// Mitsubishi GX Works2 project: C412_23-08-19 Backup   PLC: Q03UDE

PROGRAM MAIN
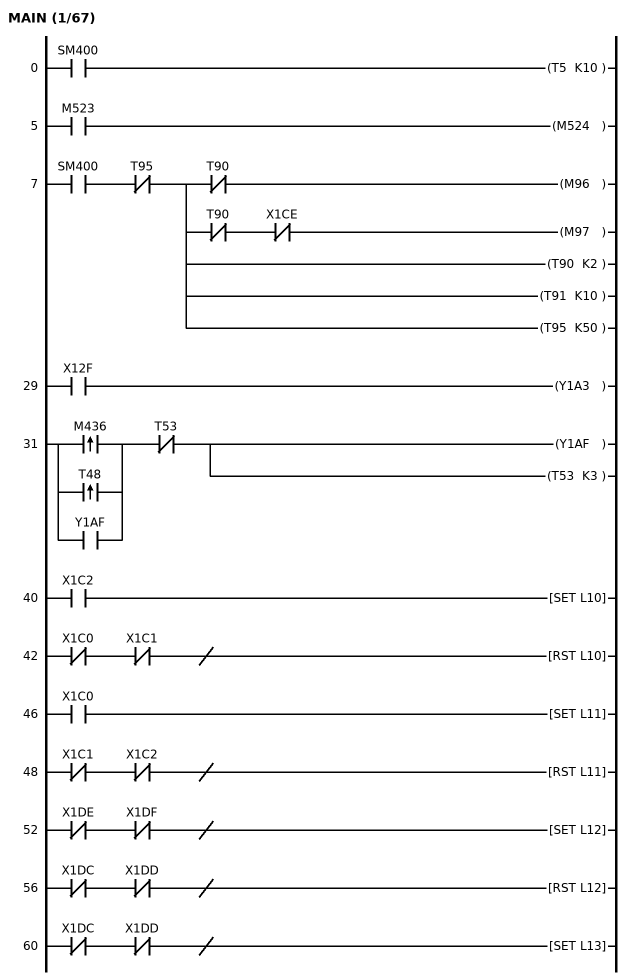
0     LD      SM400
      OUT     T5 K10
5     LD      M523
      OUT     M524
7     LD      SM400
      ANI     T95
      MPS
      ANI     T90
      OUT     M96
      MRD
      ANI     T90
      ANI     X1CE
      OUT     M97
      MPP
      OUT     T90 K2
      OUT     T91 K10
      OUT     T95 K50
29    LD      X12F
      OUT     Y1A3
31    LDP     M436
      ORP     T48
      OR      Y1AF
      ANI     T53
      OUT     Y1AF
      OUT     T53 K3
40    LD      X1C2
      SET     L10
42    LDI     X1C0
      ANI     X1C1
      INV
      RST     L10
46    LD      X1C0
      SET     L11
48    LDI     X1C1
      ANI     X1C2
      INV
      RST     L11
52    LDI     X1DE
      ANI     X1DF
      INV
      SET     L12
56    LDI     X1DC
      ANI     X1DD
      INV
      RST     L12
60    LDI     X1DC
      ANI     X1DD
      INV
      SET     L13
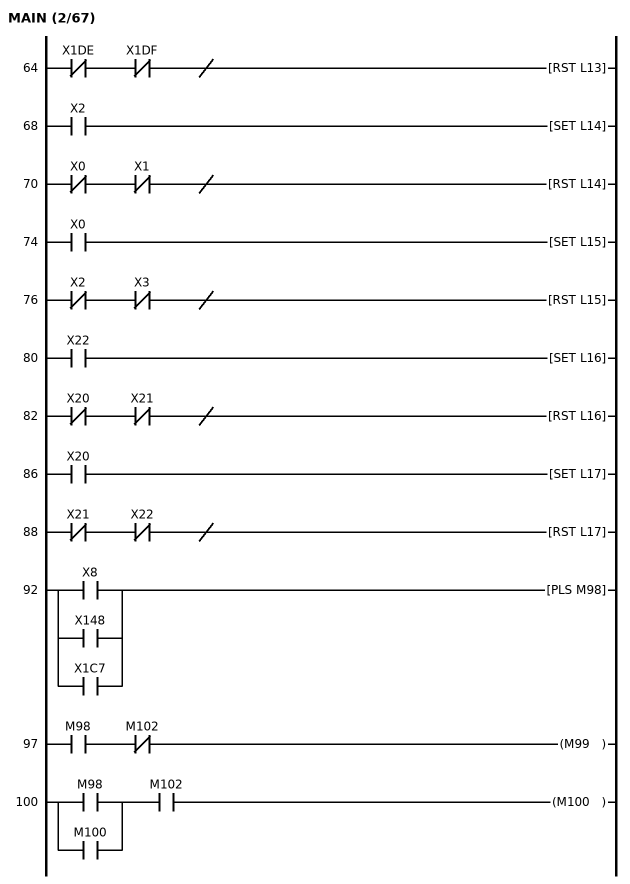
64    LDI     X1DE
      ANI     X1DF
      INV
      RST     L13
68    LD      X2
      SET     L14
70    LDI     X0
      ANI     X1
      INV
      RST     L14
74    LD      X0
      SET     L15
76    LDI     X2
      ANI     X3
      INV
      RST     L15
80    LD      X22
      SET     L16
82    LDI     X20
      ANI     X21
      INV
      RST     L16
86    LD      X20
      SET     L17
88    LDI     X21
      ANI     X22
      INV
      RST     L17
92    LD      X8
      OR      X148
      OR      X1C7
      PLS     M98
97    LD      M98
      ANI     M102
      OUT     M99
100   LD      M98
      OR      M100
      AND     M102
      OUT     M100
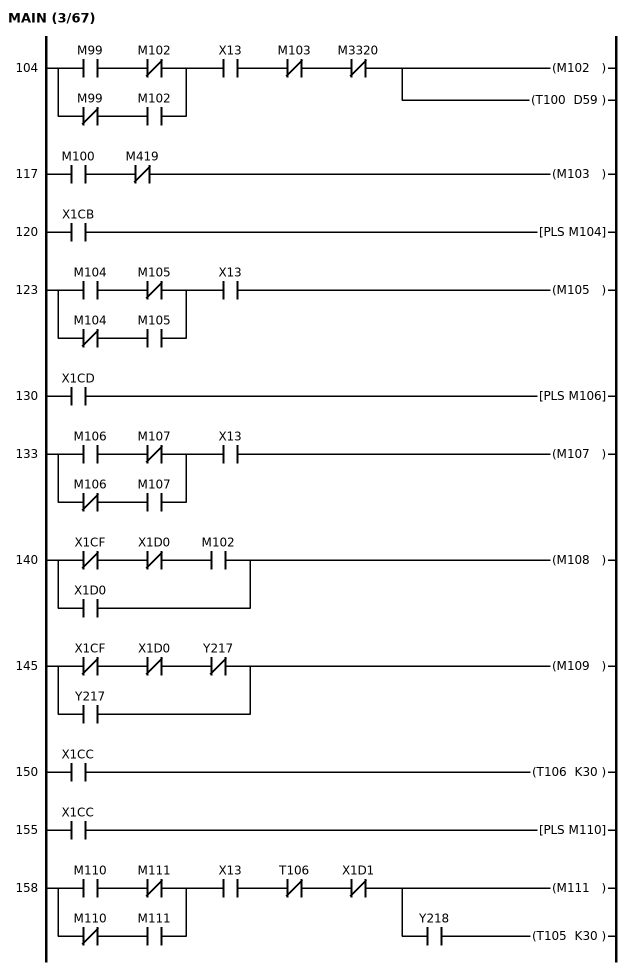
104   LD      M99
      ANI     M102
      LDI     M99
      AND     M102
      ORB
      AND     X13
      ANI     M103
      ANI     M3320
      OUT     M102
      OUT     T100 D59
117   LD      M100
      ANI     M419
      OUT     M103
120   LD      X1CB
      PLS     M104
123   LD      M104
      ANI     M105
      LDI     M104
      AND     M105
      ORB
      AND     X13
      OUT     M105
130   LD      X1CD
      PLS     M106
133   LD      M106
      ANI     M107
      LDI     M106
      AND     M107
      ORB
      AND     X13
      OUT     M107
140   LDI     X1CF
      ANI     X1D0
      AND     M102
      OR      X1D0
      OUT     M108
145   LDI     X1CF
      ANI     X1D0
      ANI     Y217
      OR      Y217
      OUT     M109
150   LD      X1CC
      OUT     T106 K30
155   LD      X1CC
      PLS     M110
158   LD      M110
      ANI     M111
      LDI     M110
      AND     M111
      ORB
      AND     X13
      ANI     T106
      ANI     X1D1
      OUT     M111
      AND     Y218
      OUT     T105 K30
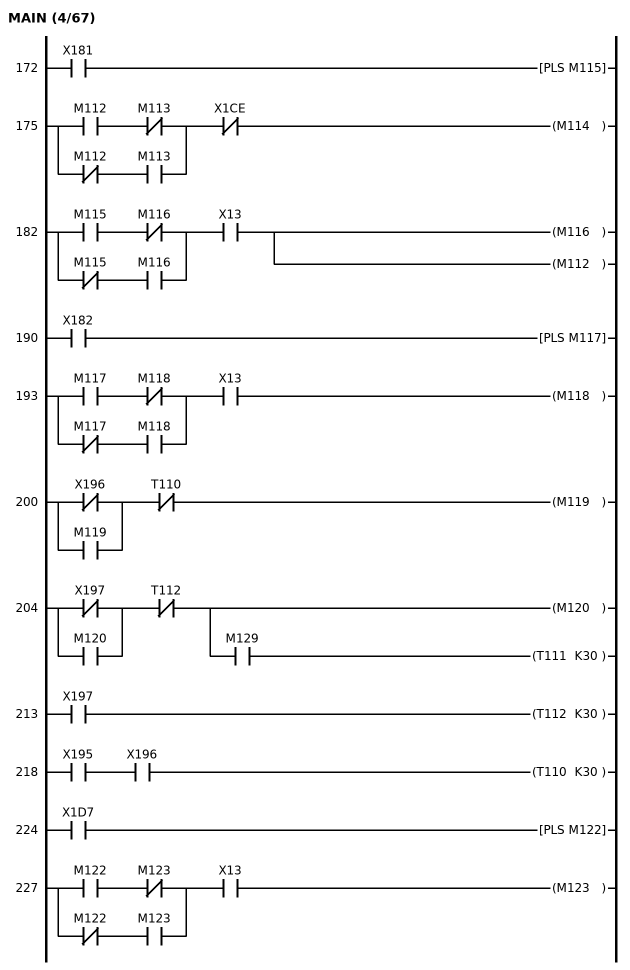
172   LD      X181
      PLS     M115
175   LD      M112
      ANI     M113
      LDI     M112
      AND     M113
      ORB
      ANI     X1CE
      OUT     M114
182   LD      M115
      ANI     M116
      LDI     M115
      AND     M116
      ORB
      AND     X13
      OUT     M116
      OUT     M112
190   LD      X182
      PLS     M117
193   LD      M117
      ANI     M118
      LDI     M117
      AND     M118
      ORB
      AND     X13
      OUT     M118
200   LDI     X196
      OR      M119
      ANI     T110
      OUT     M119
204   LDI     X197
      OR      M120
      ANI     T112
      OUT     M120
      AND     M129
      OUT     T111 K30
213   LD      X197
      OUT     T112 K30
218   LD      X195
      AND     X196
      OUT     T110 K30
224   LD      X1D7
      PLS     M122
227   LD      M122
      ANI     M123
      LDI     M122
      AND     M123
      ORB
      AND     X13
      OUT     M123
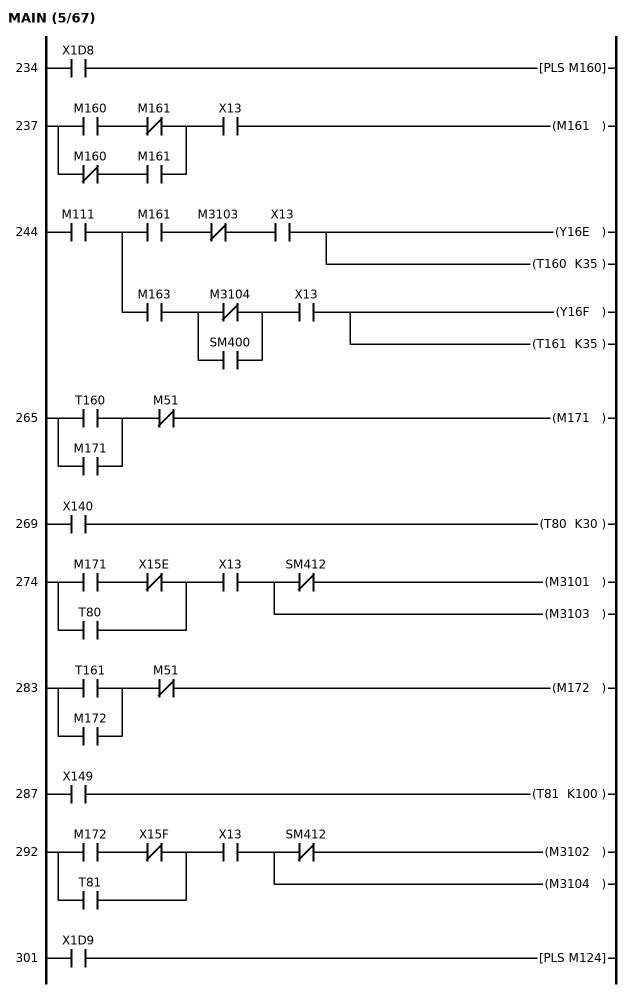
234   LD      X1D8
      PLS     M160
237   LD      M160
      ANI     M161
      LDI     M160
      AND     M161
      ORB
      AND     X13
      OUT     M161
244   LD      M111
      MPS
      AND     M161
      ANI     M3103
      AND     X13
      OUT     Y16E
      OUT     T160 K35
      MPP
      AND     M163
      LDI     M3104
      OR      SM400
      ANB
      AND     X13
      OUT     Y16F
      OUT     T161 K35
265   LD      T160
      OR      M171
      ANI     M51
      OUT     M171
269   LD      X140
      OUT     T80 K30
274   LD      M171
      ANI     X15E
      OR      T80
      AND     X13
      MPS
      ANI     SM412
      OUT     M3101
      MPP
      OUT     M3103
283   LD      T161
      OR      M172
      ANI     M51
      OUT     M172
287   LD      X149
      OUT     T81 K100
292   LD      M172
      ANI     X15F
      OR      T81
      AND     X13
      MPS
      ANI     SM412
      OUT     M3102
      MPP
      OUT     M3104
301   LD      X1D9
      PLS     M124
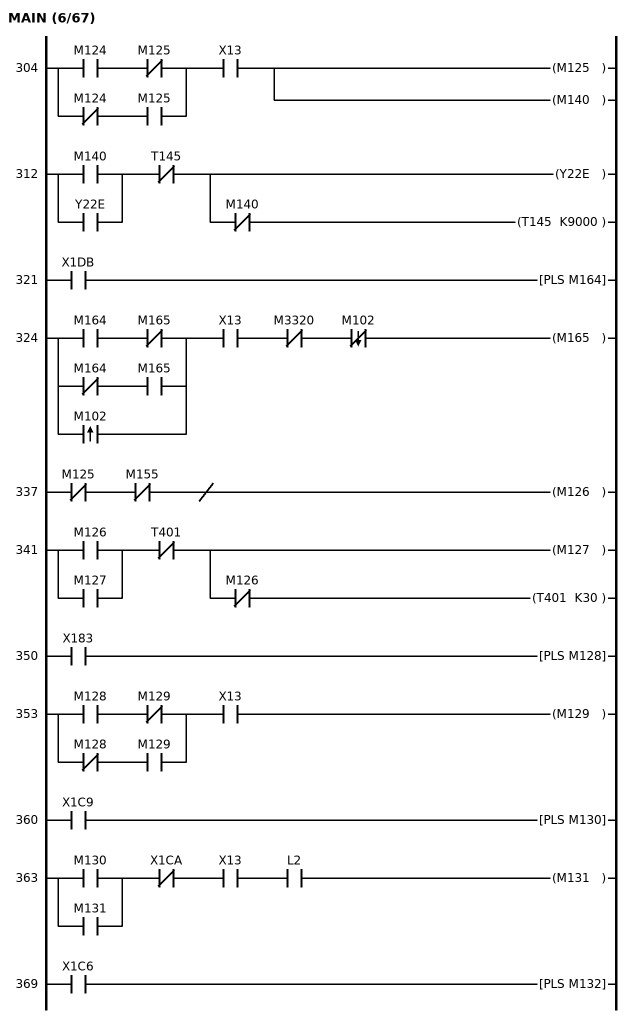
304   LD      M124
      ANI     M125
      LDI     M124
      AND     M125
      ORB
      AND     X13
      OUT     M125
      OUT     M140
312   LD      M140
      OR      Y22E
      ANI     T145
      OUT     Y22E
      ANI     M140
      OUT     T145 K9000
321   LD      X1DB
      PLS     M164
324   LD      M164
      ANI     M165
      LDI     M164
      AND     M165
      ORB
      ORP     M102
      AND     X13
      ANI     M3320
      ANDFI   M102
      OUT     M165
337   LDI     M125
      ANI     M155
      INV
      OUT     M126
341   LD      M126
      OR      M127
      ANI     T401
      OUT     M127
      ANI     M126
      OUT     T401 K30
350   LD      X183
      PLS     M128
353   LD      M128
      ANI     M129
      LDI     M128
      AND     M129
      ORB
      AND     X13
      OUT     M129
360   LD      X1C9
      PLS     M130
363   LD      M130
      OR      M131
      ANI     X1CA
      AND     X13
      AND     L2
      OUT     M131
369   LD      X1C6
      PLS     M132
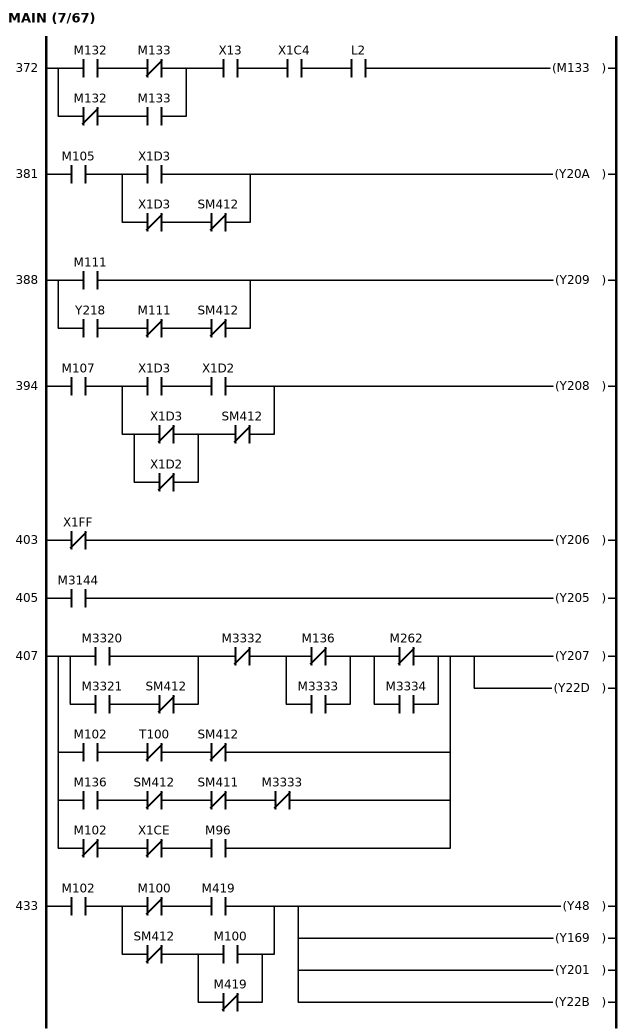
372   LD      M132
      ANI     M133
      LDI     M132
      AND     M133
      ORB
      AND     X13
      AND     X1C4
      AND     L2
      OUT     M133
381   LD      M105
      LD      X1D3
      LDI     X1D3
      ANI     SM412
      ORB
      ANB
      OUT     Y20A
388   LD      M111
      LD      Y218
      ANI     M111
      ANI     SM412
      ORB
      OUT     Y209
394   LD      M107
      LD      X1D3
      AND     X1D2
      LDI     X1D3
      ORI     X1D2
      ANI     SM412
      ORB
      ANB
      OUT     Y208
403   LDI     X1FF
      OUT     Y206
405   LD      M3144
      OUT     Y205
407   LD      M3320
      LD      M3321
      ANI     SM412
      ORB
      ANI     M3332
      LDI     M136
      OR      M3333
      ANB
      LDI     M262
      OR      M3334
      ANB
      LD      M102
      ANI     T100
      ANI     SM412
      ORB
      LD      M136
      ANI     SM412
      ANI     SM411
      ANI     M3333
      ORB
      LDI     M102
      ANI     X1CE
      AND     M96
      ORB
      OUT     Y207
      OUT     Y22D
433   LD      M102
      LDI     M100
      AND     M419
      LDI     SM412
      LD      M100
      ORI     M419
      ANB
      ORB
      ANB
      OUT     Y48
      OUT     Y169
      OUT     Y201
      OUT     Y22B
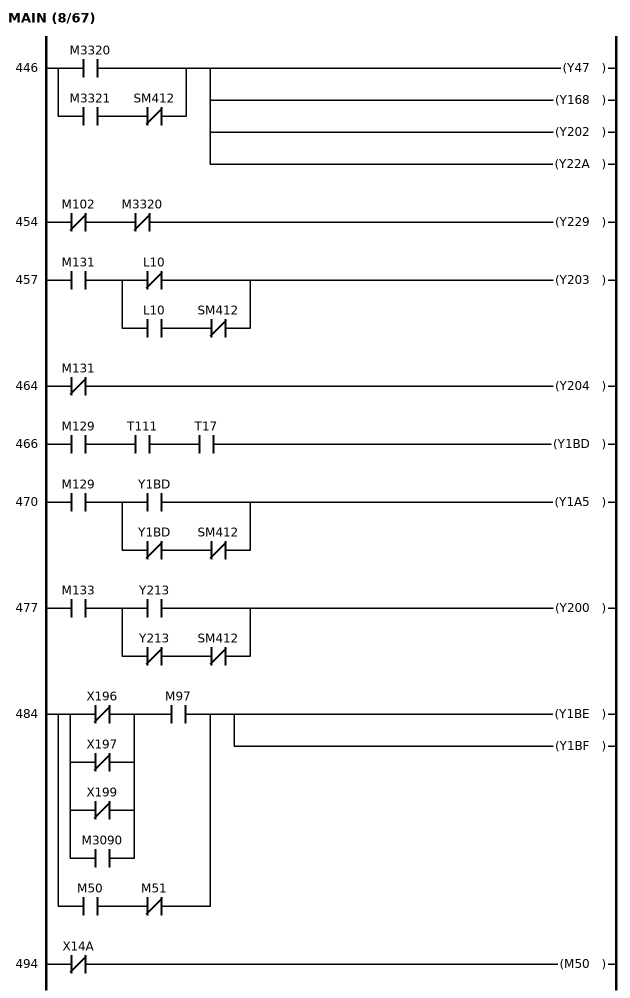
446   LD      M3320
      LD      M3321
      ANI     SM412
      ORB
      OUT     Y47
      OUT     Y168
      OUT     Y202
      OUT     Y22A
454   LDI     M102
      ANI     M3320
      OUT     Y229
457   LD      M131
      LDI     L10
      LD      L10
      ANI     SM412
      ORB
      ANB
      OUT     Y203
464   LDI     M131
      OUT     Y204
466   LD      M129
      AND     T111
      AND     T17
      OUT     Y1BD
470   LD      M129
      LD      Y1BD
      LDI     Y1BD
      ANI     SM412
      ORB
      ANB
      OUT     Y1A5
477   LD      M133
      LD      Y213
      LDI     Y213
      ANI     SM412
      ORB
      ANB
      OUT     Y200
484   LDI     X196
      ORI     X197
      ORI     X199
      OR      M3090
      AND     M97
      LD      M50
      ANI     M51
      ORB
      OUT     Y1BE
      OUT     Y1BF
494   LDI     X14A
      OUT     M50
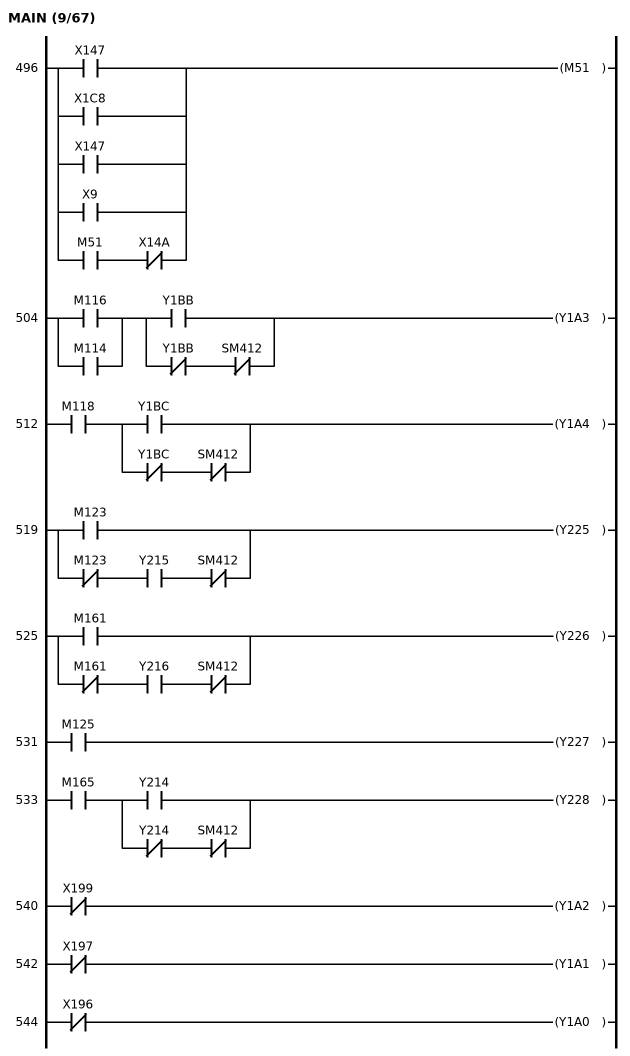
496   LD      X147
      OR      X1C8
      OR      X147
      OR      X9
      LD      M51
      ANI     X14A
      ORB
      OUT     M51
504   LD      M116
      OR      M114
      LD      Y1BB
      LDI     Y1BB
      ANI     SM412
      ORB
      ANB
      OUT     Y1A3
512   LD      M118
      LD      Y1BC
      LDI     Y1BC
      ANI     SM412
      ORB
      ANB
      OUT     Y1A4
519   LD      M123
      LDI     M123
      AND     Y215
      ANI     SM412
      ORB
      OUT     Y225
525   LD      M161
      LDI     M161
      AND     Y216
      ANI     SM412
      ORB
      OUT     Y226
531   LD      M125
      OUT     Y227
533   LD      M165
      LD      Y214
      LDI     Y214
      ANI     SM412
      ORB
      ANB
      OUT     Y228
540   LDI     X199
      OUT     Y1A2
542   LDI     X197
      OUT     Y1A1
544   LDI     X196
      OUT     Y1A0
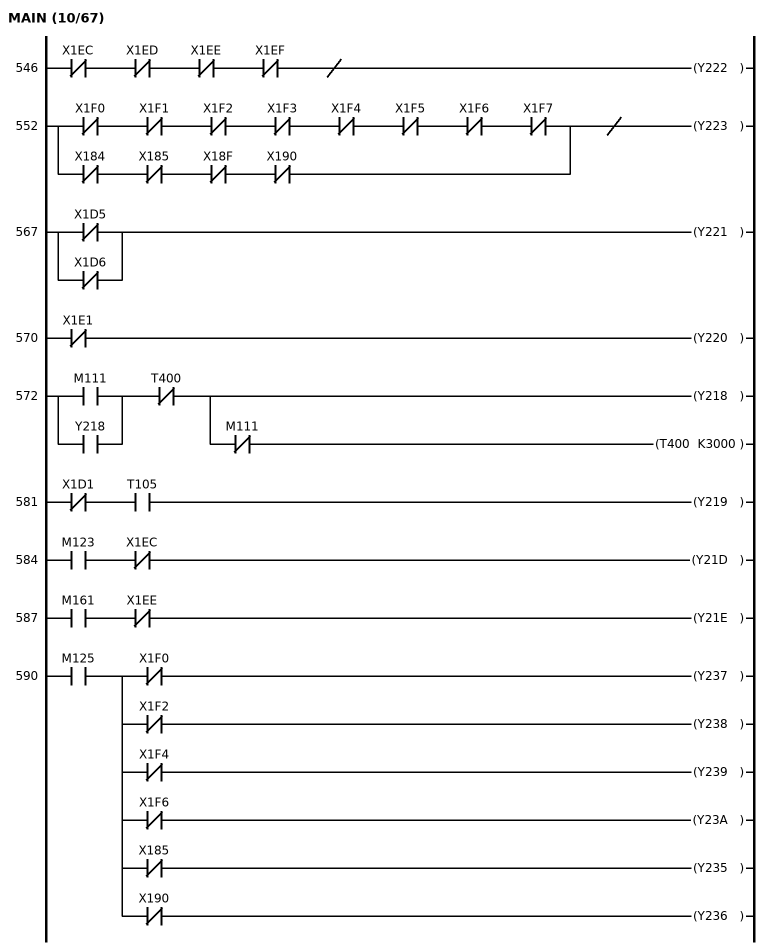
546   LDI     X1EC
      ANI     X1ED
      ANI     X1EE
      ANI     X1EF
      INV
      OUT     Y222
552   LDI     X1F0
      ANI     X1F1
      ANI     X1F2
      ANI     X1F3
      ANI     X1F4
      ANI     X1F5
      ANI     X1F6
      ANI     X1F7
      LDI     X184
      ANI     X185
      ANI     X18F
      ANI     X190
      ORB
      INV
      OUT     Y223
567   LDI     X1D5
      ORI     X1D6
      OUT     Y221
570   LDI     X1E1
      OUT     Y220
572   LD      M111
      OR      Y218
      ANI     T400
      OUT     Y218
      ANI     M111
      OUT     T400 K3000
581   LDI     X1D1
      AND     T105
      OUT     Y219
584   LD      M123
      ANI     X1EC
      OUT     Y21D
587   LD      M161
      ANI     X1EE
      OUT     Y21E
590   LD      M125
      MPS
      ANI     X1F0
      OUT     Y237
      MRD
      ANI     X1F2
      OUT     Y238
      MRD
      ANI     X1F4
      OUT     Y239
      MRD
      ANI     X1F6
      OUT     Y23A
      MRD
      ANI     X185
      OUT     Y235
      MPP
      ANI     X190
      OUT     Y236
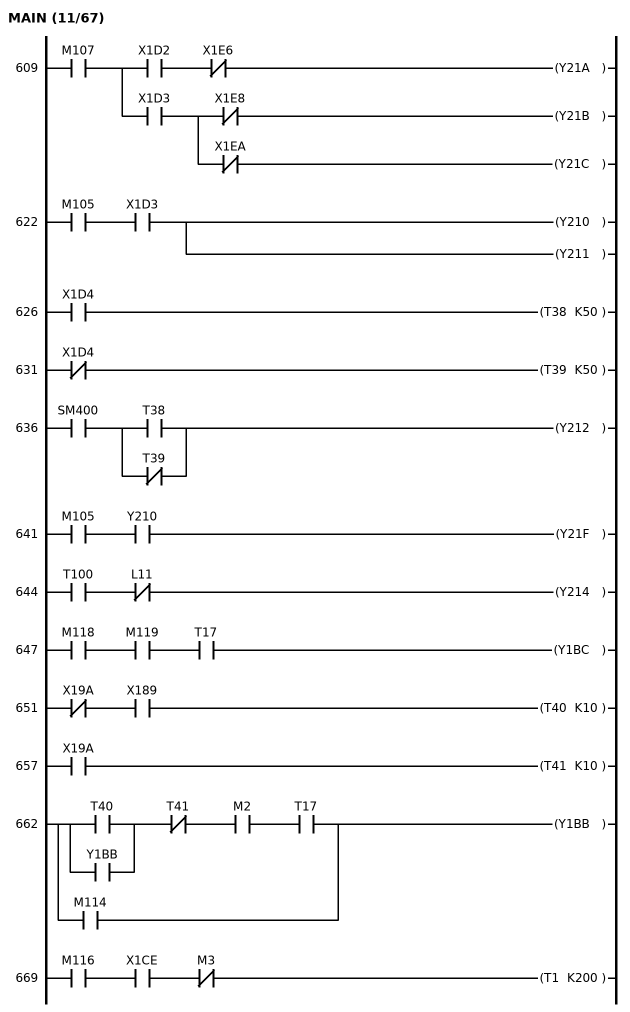
609   LD      M107
      MPS
      AND     X1D2
      ANI     X1E6
      OUT     Y21A
      MPP
      AND     X1D3
      MPS
      ANI     X1E8
      OUT     Y21B
      MPP
      ANI     X1EA
      OUT     Y21C
622   LD      M105
      AND     X1D3
      OUT     Y210
      OUT     Y211
626   LD      X1D4
      OUT     T38 K50
631   LDI     X1D4
      OUT     T39 K50
636   LD      SM400
      LD      T38
      ORI     T39
      ANB
      OUT     Y212
641   LD      M105
      AND     Y210
      OUT     Y21F
644   LD      T100
      ANI     L11
      OUT     Y214
647   LD      M118
      AND     M119
      AND     T17
      OUT     Y1BC
651   LDI     X19A
      AND     X189
      OUT     T40 K10
657   LD      X19A
      OUT     T41 K10
662   LD      T40
      OR      Y1BB
      ANI     T41
      AND     M2
      AND     T17
      OR      M114
      OUT     Y1BB
669   LD      M116
      AND     X1CE
      ANI     M3
      OUT     T1 K200
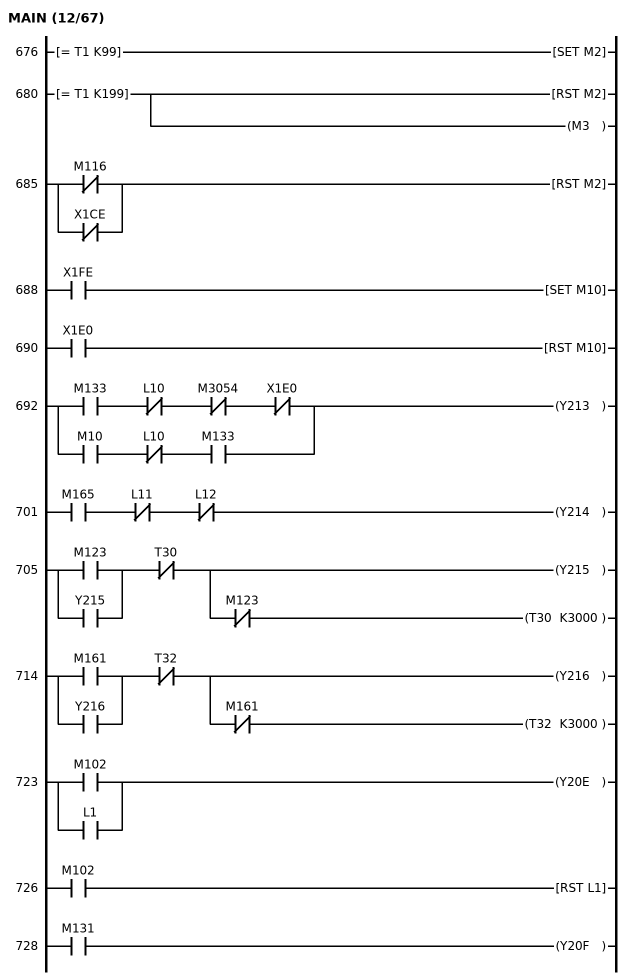
676   LD=     T1 K99
      SET     M2
680   LD=     T1 K199
      RST     M2
      OUT     M3
685   LDI     M116
      ORI     X1CE
      RST     M2
688   LD      X1FE
      SET     M10
690   LD      X1E0
      RST     M10
692   LD      M133
      ANI     L10
      ANI     M3054
      ANI     X1E0
      LD      M10
      ANI     L10
      AND     M133
      ORB
      OUT     Y213
701   LD      M165
      ANI     L11
      ANI     L12
      OUT     Y214
705   LD      M123
      OR      Y215
      ANI     T30
      OUT     Y215
      ANI     M123
      OUT     T30 K3000
714   LD      M161
      OR      Y216
      ANI     T32
      OUT     Y216
      ANI     M161
      OUT     T32 K3000
723   LD      M102
      OR      L1
      OUT     Y20E
726   LD      M102
      RST     L1
728   LD      M131
      OUT     Y20F
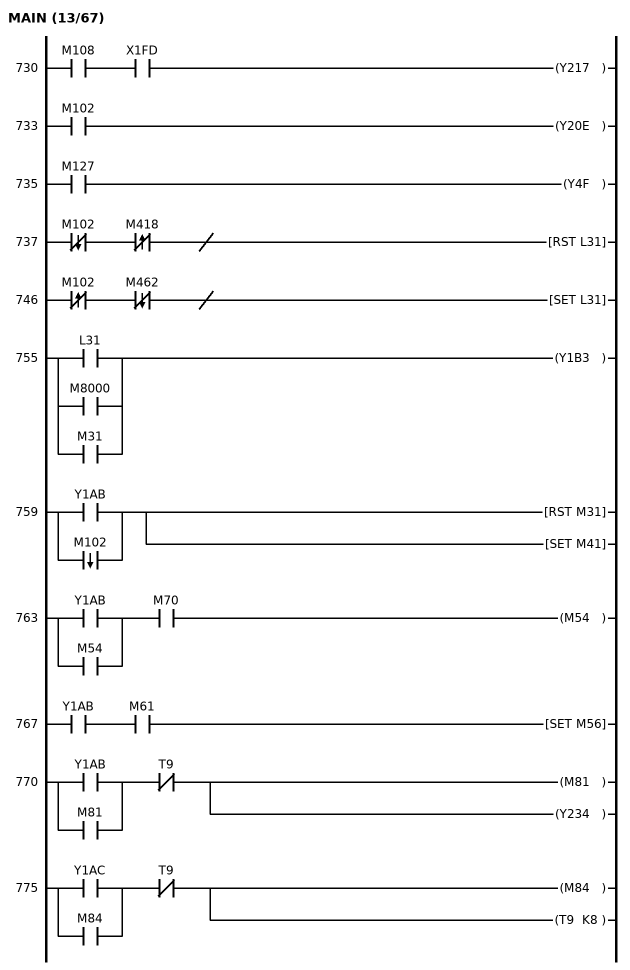
730   LD      M108
      AND     X1FD
      OUT     Y217
733   LD      M102
      OUT     Y20E
735   LD      M127
      OUT     Y4F
737   LDFI    M102
      ANDPI   M418
      INV
      RST     L31
746   LDPI    M102
      ANDFI   M462
      INV
      SET     L31
755   LD      L31
      OR      M8000
      OR      M31
      OUT     Y1B3
759   LD      Y1AB
      ORF     M102
      RST     M31
      SET     M41
763   LD      Y1AB
      OR      M54
      AND     M70
      OUT     M54
767   LD      Y1AB
      AND     M61
      SET     M56
770   LD      Y1AB
      OR      M81
      ANI     T9
      OUT     M81
      OUT     Y234
775   LD      Y1AC
      OR      M84
      ANI     T9
      OUT     M84
      OUT     T9 K8
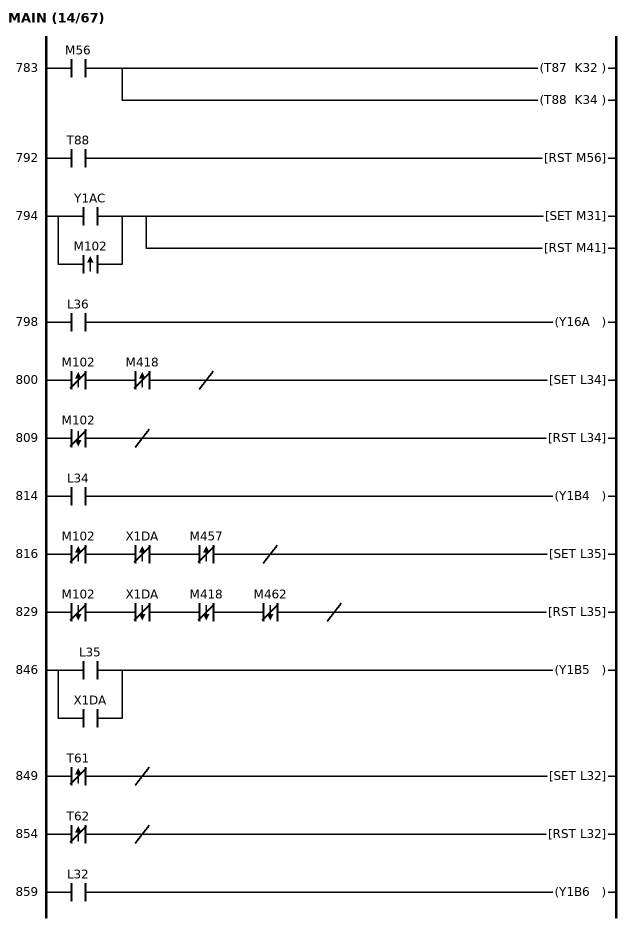
783   LD      M56
      OUT     T87 K32
      OUT     T88 K34
792   LD      T88
      RST     M56
794   LD      Y1AC
      ORP     M102
      SET     M31
      RST     M41
798   LD      L36
      OUT     Y16A
800   LDPI    M102
      ANDPI   M418
      INV
      SET     L34
809   LDFI    M102
      INV
      RST     L34
814   LD      L34
      OUT     Y1B4
816   LDPI    M102
      ANDPI   X1DA
      ANDPI   M457
      INV
      SET     L35
829   LDFI    M102
      ANDFI   X1DA
      ANDFI   M418
      ANDFI   M462
      INV
      RST     L35
846   LD      L35
      OR      X1DA
      OUT     Y1B5
849   LDPI    T61
      INV
      SET     L32
854   LDPI    T62
      INV
      RST     L32
859   LD      L32
      OUT     Y1B6
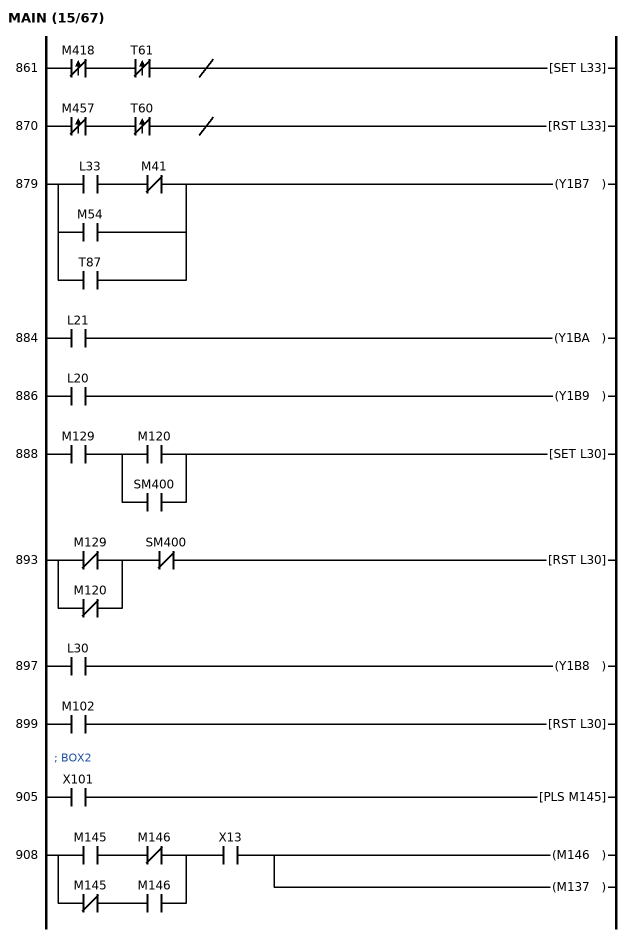
861   LDPI    M418
      ANDPI   T61
      INV
      SET     L33
870   LDPI    M457
      ANDPI   T60
      INV
      RST     L33
879   LD      L33
      ANI     M41
      OR      M54
      OR      T87
      OUT     Y1B7
884   LD      L21
      OUT     Y1BA
886   LD      L20
      OUT     Y1B9
888   LD      M129
      LD      M120
      OR      SM400
      ANB
      SET     L30
893   LDI     M129
      ORI     M120
      ANI     SM400
      RST     L30
897   LD      L30
      OUT     Y1B8
899   LD      M102
      RST     L30
; BOX2
905   LD      X101
      PLS     M145
908   LD      M145
      ANI     M146
      LDI     M145
      AND     M146
      ORB
      AND     X13
      OUT     M146
      OUT     M137
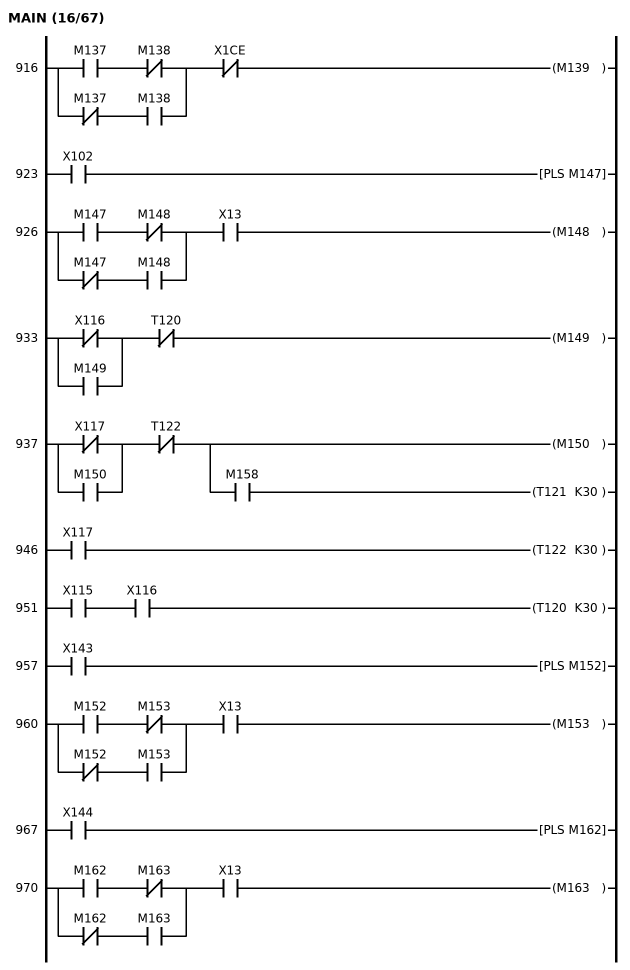
916   LD      M137
      ANI     M138
      LDI     M137
      AND     M138
      ORB
      ANI     X1CE
      OUT     M139
923   LD      X102
      PLS     M147
926   LD      M147
      ANI     M148
      LDI     M147
      AND     M148
      ORB
      AND     X13
      OUT     M148
933   LDI     X116
      OR      M149
      ANI     T120
      OUT     M149
937   LDI     X117
      OR      M150
      ANI     T122
      OUT     M150
      AND     M158
      OUT     T121 K30
946   LD      X117
      OUT     T122 K30
951   LD      X115
      AND     X116
      OUT     T120 K30
957   LD      X143
      PLS     M152
960   LD      M152
      ANI     M153
      LDI     M152
      AND     M153
      ORB
      AND     X13
      OUT     M153
967   LD      X144
      PLS     M162
970   LD      M162
      ANI     M163
      LDI     M162
      AND     M163
      ORB
      AND     X13
      OUT     M163
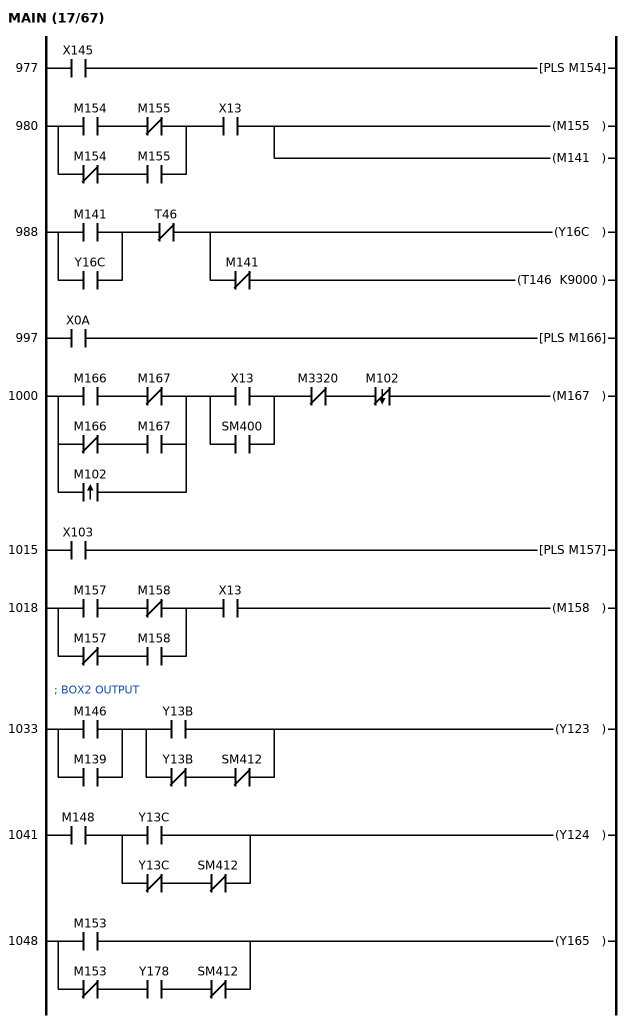
977   LD      X145
      PLS     M154
980   LD      M154
      ANI     M155
      LDI     M154
      AND     M155
      ORB
      AND     X13
      OUT     M155
      OUT     M141
988   LD      M141
      OR      Y16C
      ANI     T46
      OUT     Y16C
      ANI     M141
      OUT     T146 K9000
997   LD      X0A
      PLS     M166
1000  LD      M166
      ANI     M167
      LDI     M166
      AND     M167
      ORB
      ORP     M102
      LD      X13
      OR      SM400
      ANB
      ANI     M3320
      ANDFI   M102
      OUT     M167
1015  LD      X103
      PLS     M157
1018  LD      M157
      ANI     M158
      LDI     M157
      AND     M158
      ORB
      AND     X13
      OUT     M158
; BOX2 OUTPUT
1033  LD      M146
      OR      M139
      LD      Y13B
      LDI     Y13B
      ANI     SM412
      ORB
      ANB
      OUT     Y123
1041  LD      M148
      LD      Y13C
      LDI     Y13C
      ANI     SM412
      ORB
      ANB
      OUT     Y124
1048  LD      M153
      LDI     M153
      AND     Y178
      ANI     SM412
      ORB
      OUT     Y165
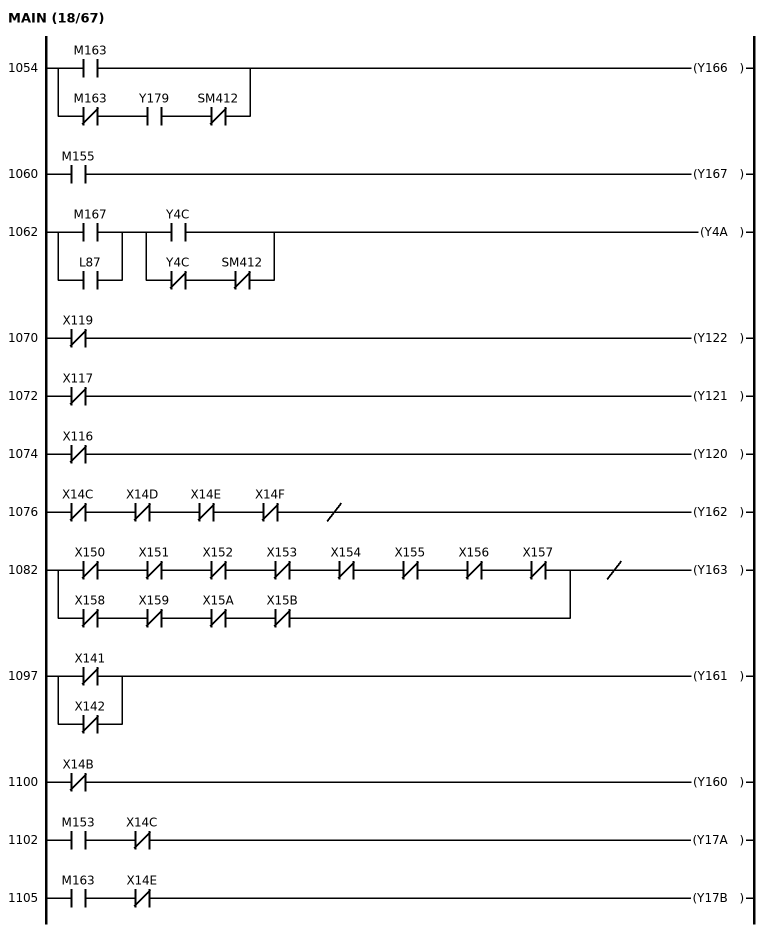
1054  LD      M163
      LDI     M163
      AND     Y179
      ANI     SM412
      ORB
      OUT     Y166
1060  LD      M155
      OUT     Y167
1062  LD      M167
      OR      L87
      LD      Y4C
      LDI     Y4C
      ANI     SM412
      ORB
      ANB
      OUT     Y4A
1070  LDI     X119
      OUT     Y122
1072  LDI     X117
      OUT     Y121
1074  LDI     X116
      OUT     Y120
1076  LDI     X14C
      ANI     X14D
      ANI     X14E
      ANI     X14F
      INV
      OUT     Y162
1082  LDI     X150
      ANI     X151
      ANI     X152
      ANI     X153
      ANI     X154
      ANI     X155
      ANI     X156
      ANI     X157
      LDI     X158
      ANI     X159
      ANI     X15A
      ANI     X15B
      ORB
      INV
      OUT     Y163
1097  LDI     X141
      ORI     X142
      OUT     Y161
1100  LDI     X14B
      OUT     Y160
1102  LD      M153
      ANI     X14C
      OUT     Y17A
1105  LD      M163
      ANI     X14E
      OUT     Y17B
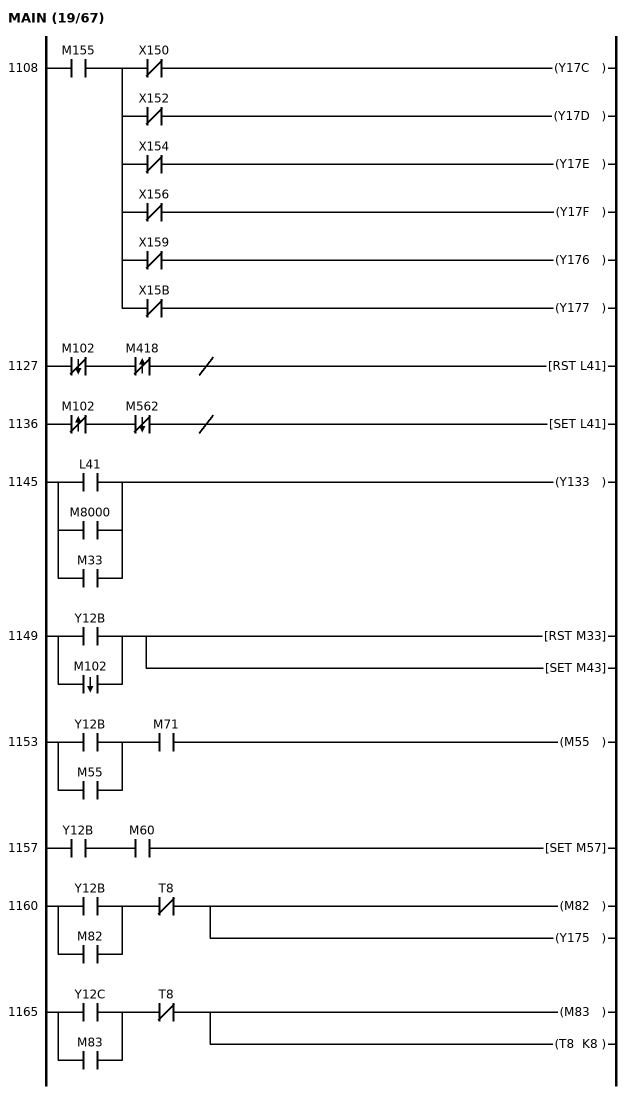
1108  LD      M155
      MPS
      ANI     X150
      OUT     Y17C
      MRD
      ANI     X152
      OUT     Y17D
      MRD
      ANI     X154
      OUT     Y17E
      MRD
      ANI     X156
      OUT     Y17F
      MRD
      ANI     X159
      OUT     Y176
      MPP
      ANI     X15B
      OUT     Y177
1127  LDFI    M102
      ANDPI   M418
      INV
      RST     L41
1136  LDPI    M102
      ANDFI   M562
      INV
      SET     L41
1145  LD      L41
      OR      M8000
      OR      M33
      OUT     Y133
1149  LD      Y12B
      ORF     M102
      RST     M33
      SET     M43
1153  LD      Y12B
      OR      M55
      AND     M71
      OUT     M55
1157  LD      Y12B
      AND     M60
      SET     M57
1160  LD      Y12B
      OR      M82
      ANI     T8
      OUT     M82
      OUT     Y175
1165  LD      Y12C
      OR      M83
      ANI     T8
      OUT     M83
      OUT     T8 K8
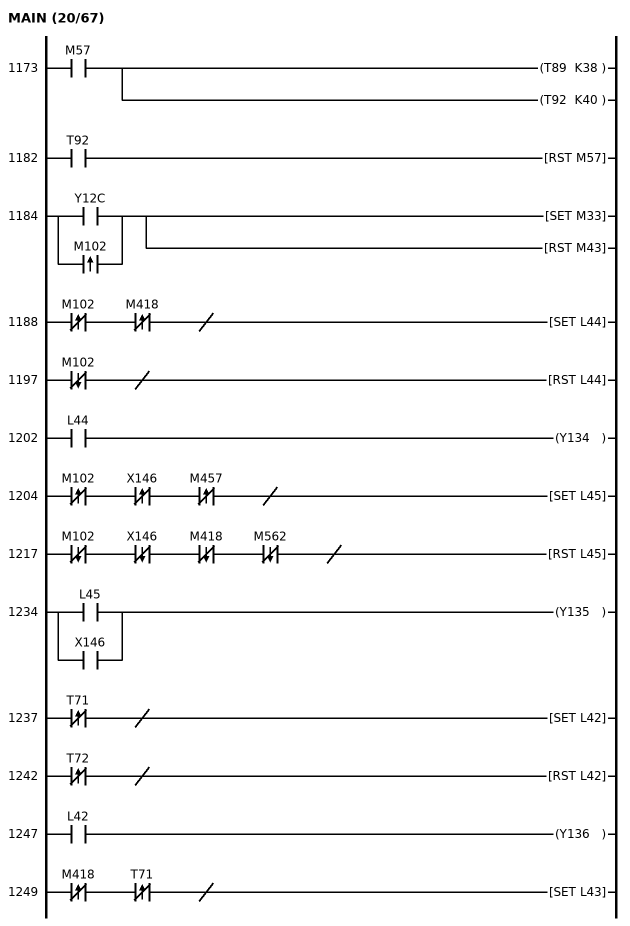
1173  LD      M57
      OUT     T89 K38
      OUT     T92 K40
1182  LD      T92
      RST     M57
1184  LD      Y12C
      ORP     M102
      SET     M33
      RST     M43
1188  LDPI    M102
      ANDPI   M418
      INV
      SET     L44
1197  LDFI    M102
      INV
      RST     L44
1202  LD      L44
      OUT     Y134
1204  LDPI    M102
      ANDPI   X146
      ANDPI   M457
      INV
      SET     L45
1217  LDFI    M102
      ANDFI   X146
      ANDFI   M418
      ANDFI   M562
      INV
      RST     L45
1234  LD      L45
      OR      X146
      OUT     Y135
1237  LDPI    T71
      INV
      SET     L42
1242  LDPI    T72
      INV
      RST     L42
1247  LD      L42
      OUT     Y136
1249  LDPI    M418
      ANDPI   T71
      INV
      SET     L43
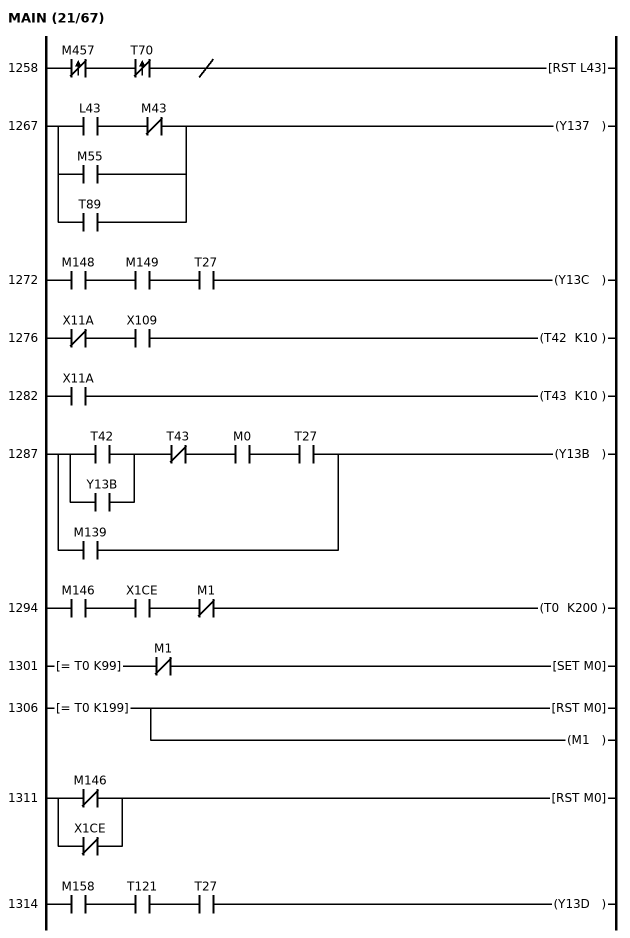
1258  LDPI    M457
      ANDPI   T70
      INV
      RST     L43
1267  LD      L43
      ANI     M43
      OR      M55
      OR      T89
      OUT     Y137
1272  LD      M148
      AND     M149
      AND     T27
      OUT     Y13C
1276  LDI     X11A
      AND     X109
      OUT     T42 K10
1282  LD      X11A
      OUT     T43 K10
1287  LD      T42
      OR      Y13B
      ANI     T43
      AND     M0
      AND     T27
      OR      M139
      OUT     Y13B
1294  LD      M146
      AND     X1CE
      ANI     M1
      OUT     T0 K200
1301  LD=     T0 K99
      ANI     M1
      SET     M0
1306  LD=     T0 K199
      RST     M0
      OUT     M1
1311  LDI     M146
      ORI     X1CE
      RST     M0
1314  LD      M158
      AND     T121
      AND     T27
      OUT     Y13D
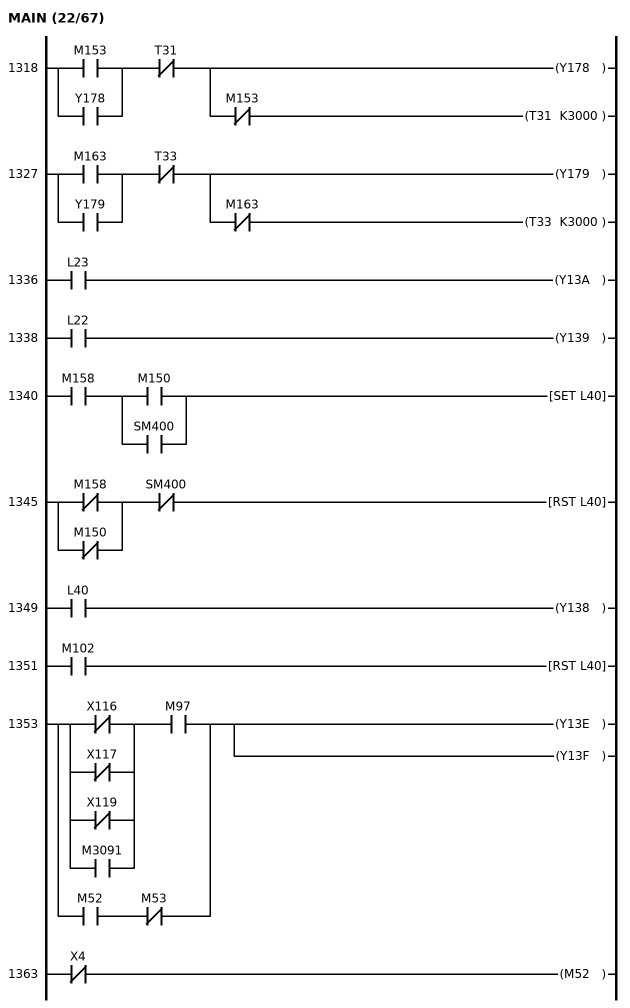
1318  LD      M153
      OR      Y178
      ANI     T31
      OUT     Y178
      ANI     M153
      OUT     T31 K3000
1327  LD      M163
      OR      Y179
      ANI     T33
      OUT     Y179
      ANI     M163
      OUT     T33 K3000
1336  LD      L23
      OUT     Y13A
1338  LD      L22
      OUT     Y139
1340  LD      M158
      LD      M150
      OR      SM400
      ANB
      SET     L40
1345  LDI     M158
      ORI     M150
      ANI     SM400
      RST     L40
1349  LD      L40
      OUT     Y138
1351  LD      M102
      RST     L40
1353  LDI     X116
      ORI     X117
      ORI     X119
      OR      M3091
      AND     M97
      LD      M52
      ANI     M53
      ORB
      OUT     Y13E
      OUT     Y13F
1363  LDI     X4
      OUT     M52
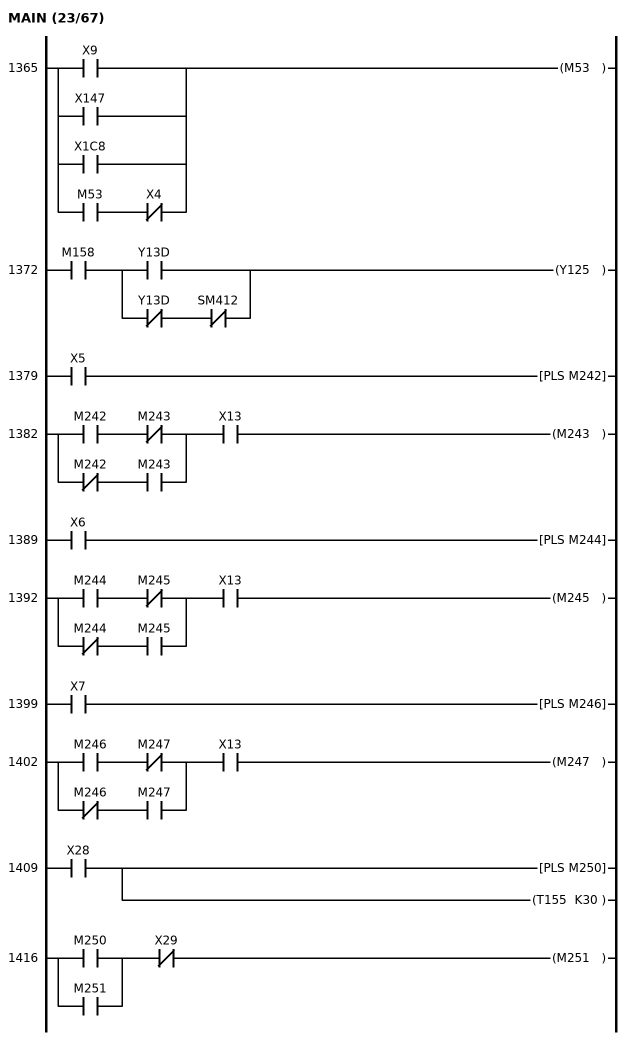
1365  LD      X9
      OR      X147
      OR      X1C8
      LD      M53
      ANI     X4
      ORB
      OUT     M53
1372  LD      M158
      LD      Y13D
      LDI     Y13D
      ANI     SM412
      ORB
      ANB
      OUT     Y125
1379  LD      X5
      PLS     M242
1382  LD      M242
      ANI     M243
      LDI     M242
      AND     M243
      ORB
      AND     X13
      OUT     M243
1389  LD      X6
      PLS     M244
1392  LD      M244
      ANI     M245
      LDI     M244
      AND     M245
      ORB
      AND     X13
      OUT     M245
1399  LD      X7
      PLS     M246
1402  LD      M246
      ANI     M247
      LDI     M246
      AND     M247
      ORB
      AND     X13
      OUT     M247
1409  LD      X28
      PLS     M250
      OUT     T155 K30
1416  LD      M250
      OR      M251
      ANI     X29
      OUT     M251
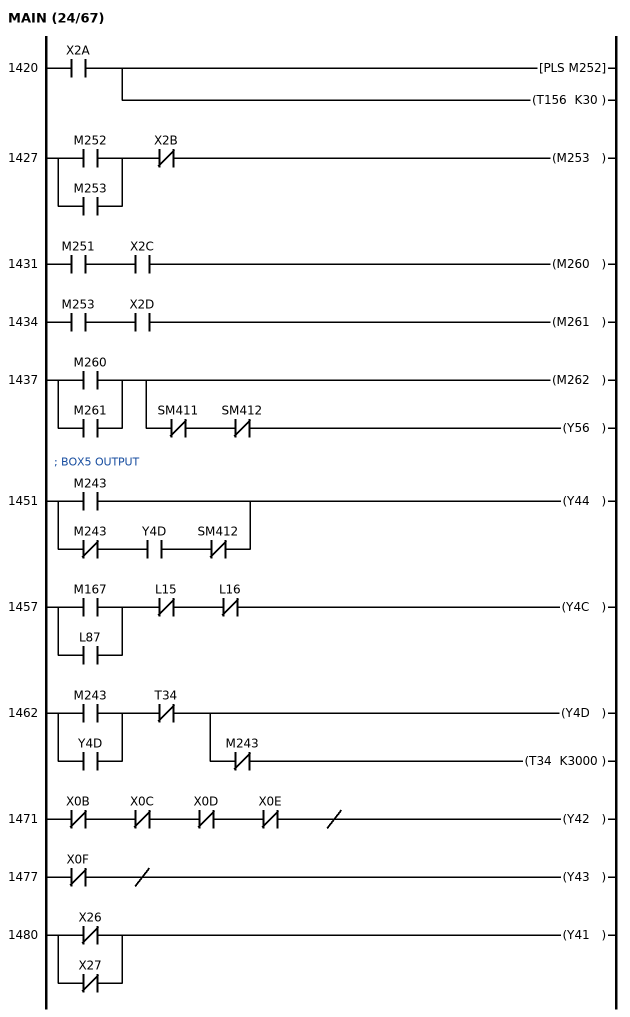
1420  LD      X2A
      PLS     M252
      OUT     T156 K30
1427  LD      M252
      OR      M253
      ANI     X2B
      OUT     M253
1431  LD      M251
      AND     X2C
      OUT     M260
1434  LD      M253
      AND     X2D
      OUT     M261
1437  LD      M260
      OR      M261
      OUT     M262
      ANI     SM411
      ANI     SM412
      OUT     Y56
; BOX5 OUTPUT
1451  LD      M243
      LDI     M243
      AND     Y4D
      ANI     SM412
      ORB
      OUT     Y44
1457  LD      M167
      OR      L87
      ANI     L15
      ANI     L16
      OUT     Y4C
1462  LD      M243
      OR      Y4D
      ANI     T34
      OUT     Y4D
      ANI     M243
      OUT     T34 K3000
1471  LDI     X0B
      ANI     X0C
      ANI     X0D
      ANI     X0E
      INV
      OUT     Y42
1477  LDI     X0F
      INV
      OUT     Y43
1480  LDI     X26
      ORI     X27
      OUT     Y41
